// Mitsubishi GX Works2 project: SET e RESET (RST) Pulsado   PLC: Q03UDV
// HelloWorld

PROGRAM MAIN
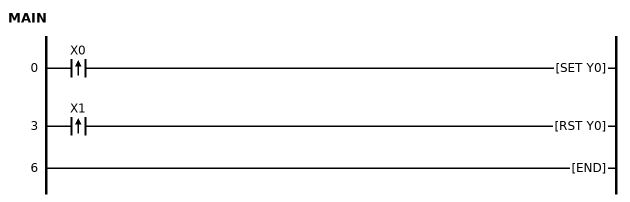
0     LDP     X0
      SET     Y0
3     LDP     X1
      RST     Y0
6     END
END_PROGRAM
